{attribute 'linkalways'} 
{attribute 'no_explicit_call' := 'This FB is a CLASS and must be accessed using methods or properties'}
{attribute 'enable_dynamic_creation'}
FUNCTION_BLOCK FINAL MUL_DINT EXTENDS Node
VAR
	in1 : _DINT(0);
	in2 : _DINT(0);
	out : _DINT(0);
END_VAR

METHOD PUBLIC Clone : I_Node
VAR
	pNode : POINTER TO MUL_DINT;
END_VAR
pNode := __NEW(MUL_DINT);
Clone := pNode^;
END_METHOD

METHOD FB_init : BOOL
VAR_INPUT
	bInitRetains : BOOL; // if TRUE, the retain variables are initialized (warm start / cold start)
	bInCopyCode : BOOL;  // if TRUE, the instance afterwards gets moved into the copy code (online change)
END_VAR
AddInput('in1',THIS^.in1);
AddInput('in2',THIS^.in2);
AddOutput('out', THIS^.out);
END_METHOD

METHOD PROTECTED OnExecute
VAR
END_VAR
out.Value := in1.Value * in2.Value;
END_METHOD

END_FUNCTION_BLOCK

(* stored: Version 1.1.0.1, ProductVersion 3.1.4024.15
   POU MUL_DINT: Id {3a0e930e-b683-43dc-aa03-340d38bace72}, SpecialFunc None
   Folder Constructor: Id {a07480fe-cee1-48d7-a591-5e50e4ac3827}
   Method Clone: Id {4c320463-8fbf-4949-b6d1-4bcfc6d50ee9}
   Method FB_init: Id {833fb6f3-165d-47c3-947c-299f0cf6d8d9}
   Method OnExecute: Id {14d0aaae-ef7e-4a5f-9c5e-c49ae784df20} *)
